// TIA Portal project "2022.04.26-计数器" (V17)

(* hardware
DEVICE "S7-1500/ET200MP station_1"  S7-1500 station
   slot 0: "导轨_0"  Rack  6ES7 590-1***0-0AA0
   slot 1: "PLC_1"  CPU 1516-3 PN/DP  6ES7 516-3AN00-0AB0  V1.7
      slot 3: "CPU 显示_1"  6ES7591-1BA00-0AA0
      slot 32768: "PROFINET 接口_1"  X1
         slot 32769: "端口_1"  X1 P1
         slot 32770: "端口_2"  X1 P2
      slot 33024: "PROFINET 接口_2"  X2
         slot 33025: "端口_1"  X2 P1
      slot 33280: "DP 接口_1"  X3
   slot 2: "DI 32x24VDC BA_1"  DI 32x24VDC BA  6ES7 521-1BL10-0AA0  V1.1
   slot 3: "DQ 32x24VDC/0.5A HF_1"  DQ 32x24VDC/0.5A HF  6ES7 522-1BL01-0AB0  V1.1
*)

// ===== PLC "PLC_1"  CPU 1516-3 PN/DP =====

VAR_GLOBAL   // PLC tag table "默认变量表"
   "按钮1" AT %I0.0 : Bool;
   "按钮2" AT %I0.1 : Bool;
   "按钮3" AT %I0.2 : Bool;
   "按钮4" AT %I0.3 : Bool;
   "按钮5" AT %I0.4 : Bool;
   "按钮6" AT %I0.5 : Bool;
   "按钮7" AT %I0.6 : Bool;
   "按钮8" AT %I0.7 : Bool;
   "按钮9" AT %I1.0 : Bool;
   "按钮10" AT %I1.1 : Bool;
   "按钮11" AT %I1.2 : Bool;
   "指示灯1" AT %Q0.0 : Bool;
   "指示灯2" AT %Q0.1 : Bool;
   "指示灯3" AT %Q0.2 : Bool;
   "指示灯4" AT %Q0.3 : Bool;
   "指示灯5" AT %Q0.4 : Bool;
   "指示灯6" AT %Q0.5 : Bool;
   "指示灯7" AT %Q0.6 : Bool;
   "指示灯8" AT %Q0.7 : Bool;
   "指示灯9" AT %Q1.0 : Bool;
   "指示灯10" AT %Q1.1 : Bool;
   "指示灯11" AT %Q1.2 : Bool;
   "指示灯12" AT %Q1.3 : Bool;
   "OLD加计数器" AT %C1 : Counter;
   "+PV" AT %MW20 : Word;
   "+CV" AT %MW22 : Word;
   "+CBD" AT %MW24 : Word;
   "-PV" AT %MW26 : Word;
   "-CV" AT %MW28 : Word;
   "-BCD" AT %MW30 : Word;
   "OLD减计数器" AT %C2 : Counter;
   "OLD+-计数器" AT %C3 : Counter;
   "OLD+-PV" AT %MW32 : Word;
   "OLD+-CV" AT %MW34 : Word;
   "OLD+-BCD" AT %MW36 : Word;
   "Tag_1" AT %C5 : Counter;
   "Tag_2" AT %C6 : Counter;
   "Tag_3" AT %C7 : Counter;
   "Tag_4" AT %C8 : Counter;
   "Tag_5" AT %C9 : Counter;
   "Tag_6" AT %C10 : Counter;
   "Tag_7" AT %C11 : Counter;
   "Tag_8" AT %C12 : Counter;
   "加计数返回值" AT %MW40 : Word;
   "减计数返回值" AT %MW42 : Int;
   "加减计数返回值" AT %MW44 : Int;
END_VAR

DATA_BLOCK "计数器LCD_DB"   // DB2
{ S7_Optimized_Access := 'TRUE' }
VERSION : 0.1
// stored: InstanceOfName 计数器LCD
"计数器LCD"
BEGIN
END_DATA_BLOCK

DATA_BLOCK "计数器FBD_DB"   // DB3
{ S7_Optimized_Access := 'TRUE' }
VERSION : 0.1
// stored: InstanceOfName 计数器FBD
"计数器FBD"
BEGIN
END_DATA_BLOCK

DATA_BLOCK "计数器LCD_DB_1"   // DB4
{ S7_Optimized_Access := 'TRUE' }
VERSION : 0.1
// stored: InstanceOfName 计数器LCD
"计数器LCD"
BEGIN
END_DATA_BLOCK

// folder: System blocks/Program resources

DATA_BLOCK "NEW加计数器"   // DB1
{ S7_Optimized_Access := 'TRUE' }
AUTHOR : Simatic
FAMILY : IEC
NAME : CNTR
VERSION : 1.0
// stored: InstanceOfName IEC_COUNTER
"IEC_COUNTER"
BEGIN
END_DATA_BLOCK

DATA_BLOCK "NEW减计数器"   // DB5
{ S7_Optimized_Access := 'TRUE' }
AUTHOR : Simatic
FAMILY : IEC
NAME : CNTR
VERSION : 1.0
// stored: InstanceOfName IEC_COUNTER
"IEC_COUNTER"
BEGIN
END_DATA_BLOCK

DATA_BLOCK "NEW加减计数器"   // DB6
{ S7_Optimized_Access := 'TRUE' }
AUTHOR : Simatic
FAMILY : IEC
NAME : CNTR
VERSION : 1.0
// stored: InstanceOfName IEC_COUNTER
"IEC_COUNTER"
BEGIN
END_DATA_BLOCK

// folder: (top level)

FUNCTION_BLOCK "计数器LCD"   // FB1, LAD
{ S7_Optimized_Access := 'TRUE' }
VERSION : 0.1
   VAR_INPUT
      Input_2 : Int;
      Input_3 : Int;
   END_VAR
   VAR RETAIN
      NEW加计数器PV : Int;
      NEW加计数器 : CTU_INT;
      NEW加计数器CV : Int;
      NEW减计数器PV : Int;
      NEW减计数器CV : Int;
      NEW减计数器 : CTD_INT;
      NEW加减计数器PV : Int;
      NEW加减计数器CV : Int;
      NEW加减计数器 : CTUD_INT;
   END_VAR
   VAR_TEMP   // added for the SCL form of the ladder/FBD networks
      _w1 : Bool;
   END_VAR
BEGIN

REGION Network 1: 加到某数亮
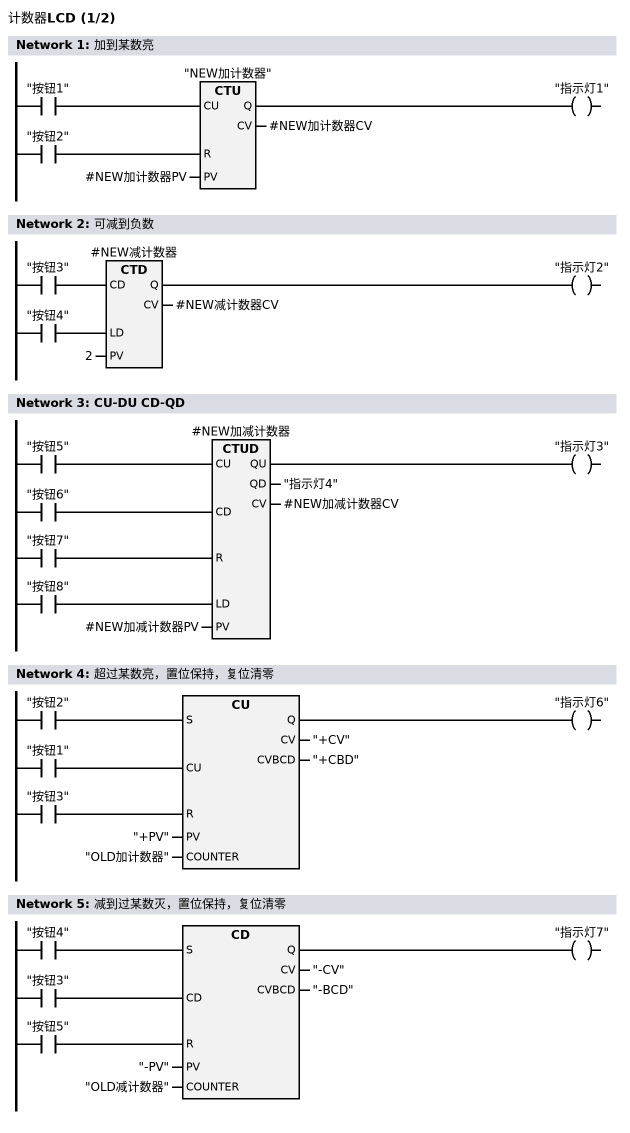
   "NEW加计数器".CTU(CU := "按钮1", R := "按钮2", PV := #NEW加计数器PV, CV => #NEW加计数器CV);
   "指示灯1" := "NEW加计数器".Q;
END_REGION

REGION Network 2: 可减到负数
   #NEW减计数器(CD := "按钮3", LD := "按钮4", PV := 2, CV => #NEW减计数器CV);   // CTD
   "指示灯2" := #NEW减计数器.Q;
END_REGION

REGION Network 3: CU-DU CD-QD
   #NEW加减计数器(CU := "按钮5",   // CTUD
             CD := "按钮6",
             R := "按钮7",
             LD := "按钮8",
             PV := #NEW加减计数器PV,
             QD => "指示灯4",
             CV => #NEW加减计数器CV);
   "指示灯3" := #NEW加减计数器.QU;
END_REGION

REGION Network 4: 超过某数亮，置位保持，复位清零
   // no SCL statement known for Cu: written as a call
   Cu(cu := "按钮1",
      s := "按钮2",
      r := "按钮3",
      pv := "+PV",
      "counter" := "OLD加计数器",
      q => #_w1,
      cv => "+CV",
      cvbcd => "+CBD");
   "指示灯6" := #_w1;
END_REGION

REGION Network 5: 减到过某数灭，置位保持，复位清零
   // no SCL statement known for Cd: written as a call
   Cd(cd := "按钮3",
      s := "按钮4",
      r := "按钮5",
      pv := "-PV",
      "counter" := "OLD减计数器",
      q => #_w1,
      cv => "-CV",
      cvbcd => "-BCD");
   "指示灯7" := #_w1;
END_REGION

REGION Network 6
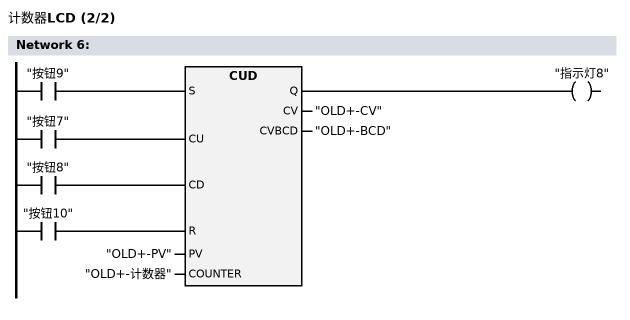
   // no SCL statement known for Cud: written as a call
   Cud(cu := "按钮7",
       cd := "按钮8",
       s := "按钮9",
       r := "按钮10",
       pv := "OLD+-PV",
       "counter" := "OLD+-计数器",
       q => #_w1,
       cv => "OLD+-CV",
       cvbcd => "OLD+-BCD");
   "指示灯8" := #_w1;
END_REGION
END_FUNCTION_BLOCK

FUNCTION_BLOCK "计数器FBD"   // FB2, FBD
{ S7_Optimized_Access := 'TRUE' }
VERSION : 0.1
   VAR RETAIN
      IEC_Counter_0_Instance : CTU_INT;
      IEC_Counter_0_Instance_1 : CTD_INT;
      IEC_Counter_0_Instance_2 : CTUD_INT;
   END_VAR
   VAR_TEMP   // added for the SCL form of the ladder/FBD networks
      _w1 : Bool;
   END_VAR
BEGIN

REGION Network 1
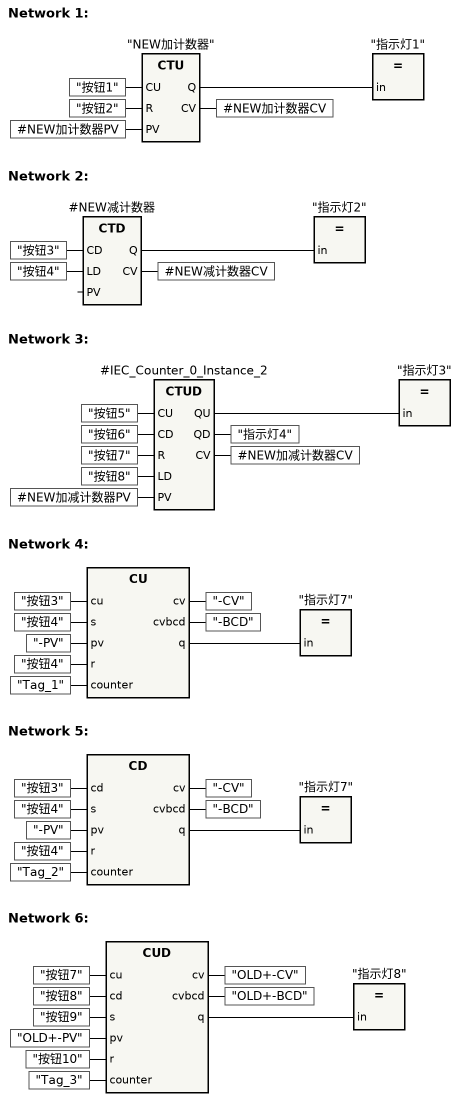
   "NEW加计数器".CTU(CU := "按钮1", R := "按钮2", PV := #NEW加计数器PV, CV => #NEW加计数器CV);
   "指示灯1" := "NEW加计数器".Q;
END_REGION

REGION Network 2
   #NEW减计数器.CTD(CD := "按钮3", LD := "按钮4", CV => #NEW减计数器CV);
   "指示灯2" := #NEW减计数器.Q;
END_REGION

REGION Network 3
   #IEC_Counter_0_Instance_2(CU := "按钮5",   // CTUD
                           CD := "按钮6",
                           R := "按钮7",
                           LD := "按钮8",
                           PV := #NEW加减计数器PV,
                           QD => "指示灯4",
                           CV => #NEW加减计数器CV);
   "指示灯3" := #IEC_Counter_0_Instance_2.QU;
END_REGION

REGION Network 4
   // no SCL statement known for Cu: written as a call
   Cu(cu := "按钮3",
      s := "按钮4",
      pv := "-PV",
      r := "按钮4",
      "counter" := "Tag_1",
      cv => "-CV",
      cvbcd => "-BCD",
      q => #_w1);
   "指示灯7" := #_w1;
END_REGION

REGION Network 5
   // no SCL statement known for Cd: written as a call
   Cd(cd := "按钮3",
      s := "按钮4",
      pv := "-PV",
      r := "按钮4",
      "counter" := "Tag_2",
      cv => "-CV",
      cvbcd => "-BCD",
      q => #_w1);
   "指示灯7" := #_w1;
END_REGION

REGION Network 6
   // no SCL statement known for Cud: written as a call
   Cud(cu := "按钮7",
       cd := "按钮8",
       s := "按钮9",
       pv := "OLD+-PV",
       r := "按钮10",
       "counter" := "Tag_3",
       cv => "OLD+-CV",
       cvbcd => "OLD+-BCD",
       q => #_w1);
   "指示灯8" := #_w1;
END_REGION
END_FUNCTION_BLOCK

FUNCTION_BLOCK "计数器SCL"   // FB3, SCL
{ S7_Optimized_Access := 'TRUE' }
VERSION : 0.1
BEGIN
   "NEW加计数器".CTU(CU:="按钮1",
                 R:="按钮2",
                 PV:=#NEW加计数器PV,
                 Q=>"指示灯1",
                 CV=>#NEW加计数器CV);

   "NEW减计数器".CTD(CD:="按钮3",
                 LD:="按钮4",
                 PV:=2,
                 Q=>"指示灯2",
                 CV=>#NEW减计数器CV);

   "NEW加减计数器".CTUD(CU:="按钮5",
                   CD:="按钮6",
                   R:="按钮7",
                   LD:="按钮8",
                   PV:=#NEW加减计数器PV,
                   QU=>"指示灯3",
                   QD=>"指示灯4",
                   CV=>#NEW加减计数器CV);

   "加计数返回值" := S_CU(C_NO := "Tag_5",
                    CU := "按钮1",
                    S := "按钮2",
                    PV := "+PV",
                    R := "按钮3",
                    CV => "+CV",
                    Q => "指示灯6");

   "减计数返回值" := S_CD(C_NO := "Tag_6",
                    CD := "按钮3",
                    S := "按钮4",
                    PV := 2,
                    R := "按钮5",
                    CV => "-CV",
                    Q => "指示灯7");

   "加减计数返回值" := S_CUD(C_NO := "Tag_7",
                      CD := "按钮8",
                      CU := "按钮7",
                      S := "按钮4",
                      PV := "OLD+-PV",
                      R := "按钮10",
                      CV => "OLD+-CV",
                      Q => "指示灯8");
END_FUNCTION_BLOCK

ORGANIZATION_BLOCK "Main"   // OB1, LAD, ProgramCycle
TITLE = "Main Program Sweep (Cycle)"
{ S7_Optimized_Access := 'TRUE' }
VERSION : 0.1
   VAR_INPUT
      Initial_Call : Bool;   // Initial call of this OB
      Remanence : Bool;   // =True, if remanent data are available
   END_VAR
BEGIN

REGION Network 1: 1
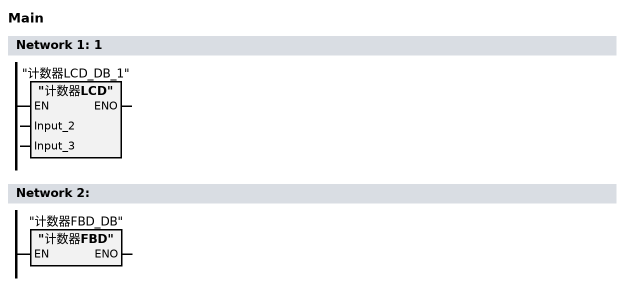
   RUNG wire#powerrail
      "计数器LCD_DB_1"(Input_2 :=, Input_3 :=)
   END_RUNG
   // the same network as SCL:
   "计数器LCD_DB_1"();   // "计数器LCD"
END_REGION

REGION Network 2
   RUNG wire#powerrail
      "计数器FBD_DB"()
   END_RUNG
   // the same network as SCL:
   "计数器FBD_DB"();   // "计数器FBD"
END_REGION
END_ORGANIZATION_BLOCK